FUNCTION BOOLS_TO_ST08B
  (* Standard: 61499-1 *)
  (* Version 1.0, 2024-02-22, franz *)
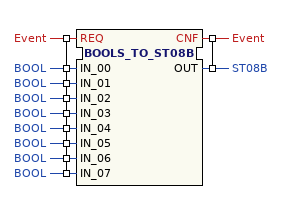
  EVENT_INPUT
    REQ WITH IN_00, IN_01, IN_02, IN_03, IN_04, IN_05, IN_06, IN_07; (* Normal Execution Request *)
  END_EVENT
  EVENT_OUTPUT
    CNF WITH OUT; (* Execution Confirmation *)
  END_EVENT
  VAR_INPUT
    IN_00 : BOOL; (* BIT 00 *)
    IN_01 : BOOL; (* BIT 01 *)
    IN_02 : BOOL; (* BIT 02 *)
    IN_03 : BOOL; (* BIT 03 *)
    IN_04 : BOOL; (* BIT 04 *)
    IN_05 : BOOL; (* BIT 05 *)
    IN_06 : BOOL; (* BIT 06 *)
    IN_07 : BOOL; (* BIT 07 *)
  END_VAR
  VAR_OUTPUT
    OUT : ST08B; (* ST08B Output *)
  END_VAR
  BODY IN ST:
FUNCTION BOOLS_TO_ST08B

VAR_INPUT
	IN_00 : BOOL;    // BIT 00
	IN_01 : BOOL;    // BIT 01
	IN_02 : BOOL;    // BIT 02
	IN_03 : BOOL;    // BIT 03
	IN_04 : BOOL;    // BIT 04
	IN_05 : BOOL;    // BIT 05
	IN_06 : BOOL;    // BIT 06
	IN_07 : BOOL;    // BIT 07
END_VAR

VAR_OUTPUT
	OUT : ST08B;    // ST08B Output
END_VAR

(* this Function extracts the 8 BOOLS from a byte *)
OUT.B_00 := IN_00;
OUT.B_01 := IN_01;
OUT.B_02 := IN_02;
OUT.B_03 := IN_03;
OUT.B_04 := IN_04;
OUT.B_05 := IN_05;
OUT.B_06 := IN_06;
OUT.B_07 := IN_07;

END_FUNCTION
  END_BODY
END_FUNCTION
